(* PLC project Addition_CFC, IEC61131-3 LD Demo Project CFC Addition Example 1.0 *)
(* stored: creationDateTime 2026-01-18T00:00:00, contentDescription CFC连续功能图加法示例程序 - 教学演示用, modificationDateTime 2026-01-18T00:00:00 *)

(* <h2>CFC连续功能图加法示例程序</h2> <p><strong>功能</strong>：实现两个INT类型整数的加法运算</p> <p><strong>编程语言</strong>：CFC（Continuous Function Chart，连续功能图）</p> <h3>变量</h3> <ul> <li>A (INT)：加数1，范围 -32768 到 32767</li> <li>B (INT)：加数2，范围 -32768 到 32767</li> <li>Result (INT)：和，存储计算结果</li> </ul> <h3>逻辑</h3> <p>使用标准ADD功能块实现 Result = A + B</p> <p>数据流：A → ADD.IN1, B → ADD.IN2, ADD.OUT → Result</p> <h3>CFC与LD的对比</h3> <ul> <li><strong>LD（梯形图）</strong>：类似继电器逻辑，从左到右、从上到下扫描</li> <li><strong>CFC（功能图）</strong>：可视化数据流，功能块可自由布局</li> <li><strong>适用场景</strong>：CFC更适合复杂算术运算和控制算法</li> </ul> <h3>测试用例</h3> <p>参见 examples/cfc/test-cases.json</p> <h3>使用指南</h3> <p>参见 examples/cfc/addition.md</p> *)
PROGRAM Addition_CFC
  VAR
    A : INT;  (* 加数1：INT类型（16位有符号整数），范围 -32768 到 32767 *)
    B : INT;  (* 加数2：INT类型（16位有符号整数），范围 -32768 到 32767 *)
    Result : INT;  (* 和：存储A + B的计算结果（INT类型，可能发生溢出回绕） *)
  END_VAR

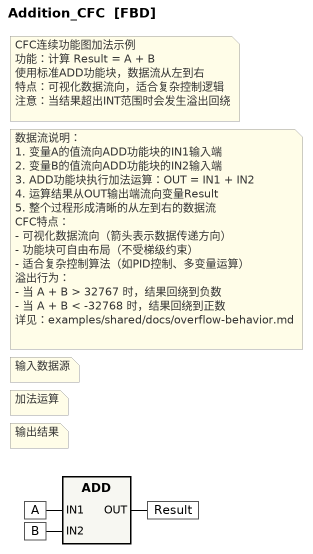
(* FBD diagram, written out as Structured Text *)
(* CFC连续功能图加法示例
                  功能：计算 Result = A + B
                  使用标准ADD功能块，数据流从左到右
                  特点：可视化数据流向，适合复杂控制逻辑
                  注意：当结果超出INT范围时会发生溢出回绕 *)
(* 加法运算 *)
(* 输入数据源 *)
(* 输出结果 *)
Result := A + B;
(* 数据流说明：
                  1. 变量A的值流向ADD功能块的IN1输入端
                  2. 变量B的值流向ADD功能块的IN2输入端
                  3. ADD功能块执行加法运算：OUT = IN1 + IN2
                  4. 运算结果从OUT输出端流向变量Result
                  5. 整个过程形成清晰的从左到右的数据流

                  CFC特点：
                  - 可视化数据流向（箭头表示数据传递方向）
                  - 功能块可自由布局（不受梯级约束）
                  - 适合复杂控制算法（如PID控制、多变量运算）

                  溢出行为：
                  - 当 A + B > 32767 时，结果回绕到负数
                  - 当 A + B < -32768 时，结果回绕到正数
                  详见：examples/shared/docs/overflow-behavior.md *)
END_PROGRAM

CONFIGURATION Config
  RESOURCE Resource1 ON PLC
    TASK MainTask(INTERVAL := T#100ms, PRIORITY := 0);
    PROGRAM Addition_CFC_Instance WITH MainTask : Addition_CFC;
  END_RESOURCE
END_CONFIGURATION
